(* PLC project time_management, Dassault Systèmes ControlBuild 2024x *)
(* stored: creationDateTime 2023-10-03T11:13:47-01:00 *)

FUNCTION_BLOCK tni_clock.time_management
  VAR_INPUT
    tick : BOOL := false;
  END_VAR
  VAR_IN_OUT
    B1 : BOOL := false;
    B2 : BOOL := false;
    B3 : BOOL := false;
    B4 : BOOL := false;
  END_VAR
  VAR_OUTPUT
    stepMotorSecond : BOOL := false;
    stepMotorMinute : BOOL := false;
    stepMotorHour : BOOL := false;
  END_VAR
  VAR_OUTPUT
    hh : SINT := 0;
    mn : SINT := 0;
    sec : SINT := 0;
  END_VAR
  VAR
    tickCount : REAL := 0.0;
    adjustMode : INT := 0;
  END_VAR

(**************   Time setting  *****************)
(* First B1 push : hour stting      *)
(* Second B1 push : minutes setting	*)
(* Third B1 push : seconds setting   *)
(* Push on B2 : current value modification       *)
(**************************************************)


(***** Motors running orders initialisation *****)
stepMotorSecond:= FALSE;
stepMotorMinute := FALSE;
stepMotorHour := FALSE;

IF (B1 OR (adjustMode > 0)) THEN
	IF B1 THEN adjustMode := adjustMode + 1; END_IF;
	B1 := FALSE;
	IF adjustMode > 3 THEN adjustMode := 0; END_IF;
	IF B2 THEN
		B2 := FALSE;
		CASE adjustMode OF
			1 : 	hh := hh + 1;
				stepMotorHour := true;	
			2 : 	mn := mn + 1;
				stepMotorMinute := true;	
			3 : 	sec := sec + 1;
				stepMotorSecond:= true;	
		END_CASE;
	END_IF;	
END_IF;

(***** Take quartz from pulse into account  ******)
(** The pulse is not take into account when setting mode is on **)
IF (RE tick and (adjustMode = 0)) THEN
	tickCount := tickCount + (CLOCK_PERIOD * 2.0); (* un RE de tick tous les 2 cycles *)
	IF tickCount > 1000000.0 THEN
		sec := sec + 1;
		stepMotorSecond := true;
		tickCount := tickCount - 1000000.0;
	END_IF;
END_IF;



(***** Current time calculation ******)	

IF sec > 60 THEN
	sec := 0;
	IF adjustMode = 0 THEN 
		mn := mn + 1;
		stepMotorMinute := true;
	END_IF;
END_IF;
IF mn > 60 THEN
	mn := 0;
	IF adjustMode = 0 THEN
		hh := hh + 1; 
		stepMotorHour := true;
	END_IF;
END_IF;
IF hh > 23 THEN
	hh := 0;	
END_IF;
END_FUNCTION_BLOCK
